Staubli VAL3: releaseSample.pgx

program releaseSample()
begin
  currentSamPosJ=herej()
  currentSamPos=jointToPoint(flange,world,currentSamPosJ)
  movel(appro(currentSamPos,{0,0,80,0,0,0}),flange,mNomSpeed)
  waitEndMove()
  switchGripper=false
  movel(appro(currentSamPos,{0,0,0,0,0,0}),flange,mNomSpeed)
  waitEndMove()
  message="releaseSample:done"
  taskCreate "sendStatus",100,sendStatus()
  taskKill ("releaseSample")
end
